{attribute addProperty BoxType "AX8206-0000-0100-0100"}
{attribute addProperty Id "Ch_B_Position_actual_value_invalidAT %I*BOOL812Ch_B_1st_Additional_position_actual_value_invalidAT %I*BOOL813Ch_B_StatuswordAT %I*UINT1620Ch_B_Position_actual_valueAT %I*DINT3240"}
{attribute addProperty CRC "3618948210"}
{attribute addProperty SizeInBites "64"}
{attribute addProperty SizeInBytes "8"}
TYPE Ch_B_AxisMain_Inputs_D7B4C472 :
STRUCT
	{attribute addProperty Name "Ch_B_Position_actual_value_invalid"}
	Ch_B_Position_actual_value_invalid AT %I* : BOOL;
	{attribute addProperty Name "Ch_B_1st_Additional_position_actual_value_invalid"}
	Ch_B_1st_Additional_position_actual_value_invalid AT %I* : BOOL;
	{attribute addProperty Name "Ch_B_Statusword"}
	Ch_B_Statusword AT %I* : UINT;
	{attribute addProperty Name "Ch_B_Position_actual_value"}
	Ch_B_Position_actual_value AT %I* : DINT;
END_STRUCT
END_TYPE

(* stored: Version 1.2.0.0, ProductVersion 3.1.4024.9
   DUT Ch_B_AxisMain_Inputs_D7B4C472: Id {24c164f5-0637-4bbe-890d-aa43d2a90a46} *)
